(* PLC project  *)

CONFIGURATION Empty_Module_8
END_CONFIGURATION
